// TIA Portal project "Fish Feeding System" (V17)
// The system should dispense 3 types of food for 5 sec every 15 sec. It will dispense food only if there is movement of fishes in the near water.

(* hardware
DEVICE "S7-1200 station_1"  S7-1200 Station
   slot 0: "Rack_0"  S7-1200 Rack  Rack  V1.0
   slot 1: "PLC_1"  CPU 1211C AC/DC/Rly  6ES7 211-1BE40-0XB0  V4.5
*)

// ===== PLC "PLC_1"  CPU 1211C AC/DC/Rly =====

VAR_GLOBAL   // PLC tag table "Default tag table"
   "Start_button" AT %I0.0 : Bool;
   "Sensor" AT %I0.1 : Bool;
   "Valve_1" AT %Q0.0 : Bool;
   "Valve_2" AT %Q0.1 : Bool;
   "Valve_3" AT %Q0.2 : Bool;
   "Tag_1" AT %M0.0 : Bool;
   "Tag_2" AT %M0.1 : Bool;
END_VAR

// folder: System blocks/Program resources

DATA_BLOCK "IEC_Timer_0_DB"   // DB1
{ S7_Optimized_Access := 'TRUE' }
AUTHOR : Simatic
FAMILY : IEC
NAME : IEC_TMR
VERSION : 1.0
// stored: InstanceOfName IEC_TIMER
"IEC_TIMER"
BEGIN
END_DATA_BLOCK

DATA_BLOCK "IEC_Timer_0_DB_1"   // DB2
{ S7_Optimized_Access := 'TRUE' }
AUTHOR : Simatic
FAMILY : IEC
NAME : IEC_TMR
VERSION : 1.0
// stored: InstanceOfName IEC_TIMER
"IEC_TIMER"
BEGIN
END_DATA_BLOCK

DATA_BLOCK "IEC_Timer_0_DB_2"   // DB3
{ S7_Optimized_Access := 'TRUE' }
AUTHOR : Simatic
FAMILY : IEC
NAME : IEC_TMR
VERSION : 1.0
// stored: InstanceOfName IEC_TIMER
"IEC_TIMER"
BEGIN
END_DATA_BLOCK

DATA_BLOCK "IEC_Timer_0_DB_3"   // DB4
{ S7_Optimized_Access := 'TRUE' }
AUTHOR : Simatic
FAMILY : IEC
NAME : IEC_TMR
VERSION : 1.0
// stored: InstanceOfName IEC_TIMER
"IEC_TIMER"
BEGIN
END_DATA_BLOCK

// folder: (top level)

ORGANIZATION_BLOCK "Main"   // OB1, LAD, ProgramCycle
TITLE = "Main Program Sweep (Cycle)"
{ S7_Optimized_Access := 'TRUE' }
VERSION : 0.1
   VAR_INPUT
      Initial_Call : Bool;   // Initial call of this OB
      Remanence : Bool;   // =True, if remanent data are available
   END_VAR
BEGIN

REGION Network 1
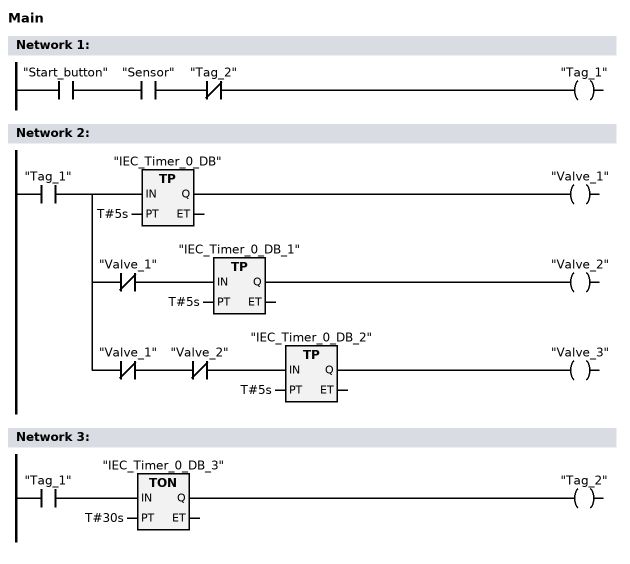
   RUNG wire#powerrail
      Contact( "Start_button" )
      Contact( "Sensor" )
      I_Contact( "Tag_2" )
      Coil( "Tag_1" )
   END_RUNG
   // the same network as SCL:
   "Tag_1" := "Start_button" AND "Sensor" AND NOT "Tag_2";
END_REGION

REGION Network 2
   "IEC_Timer_0_DB".TP(IN := "Tag_1", PT := T#5s);
   "Valve_1" := "IEC_Timer_0_DB".Q;
   "IEC_Timer_0_DB_1".TP(IN := "Tag_1" AND NOT "Valve_1", PT := T#5s);
   "Valve_2" := "IEC_Timer_0_DB_1".Q;
   "IEC_Timer_0_DB_2".TP(IN := "Tag_1" AND NOT "Valve_1" AND NOT "Valve_2", PT := T#5s);
   "Valve_3" := "IEC_Timer_0_DB_2".Q;
END_REGION

REGION Network 3
   "IEC_Timer_0_DB_3".TON(IN := "Tag_1", PT := T#30s);
   "Tag_2" := "IEC_Timer_0_DB_3".Q;
END_REGION
END_ORGANIZATION_BLOCK